RoboDK station: SandBox_RS003N.rdk

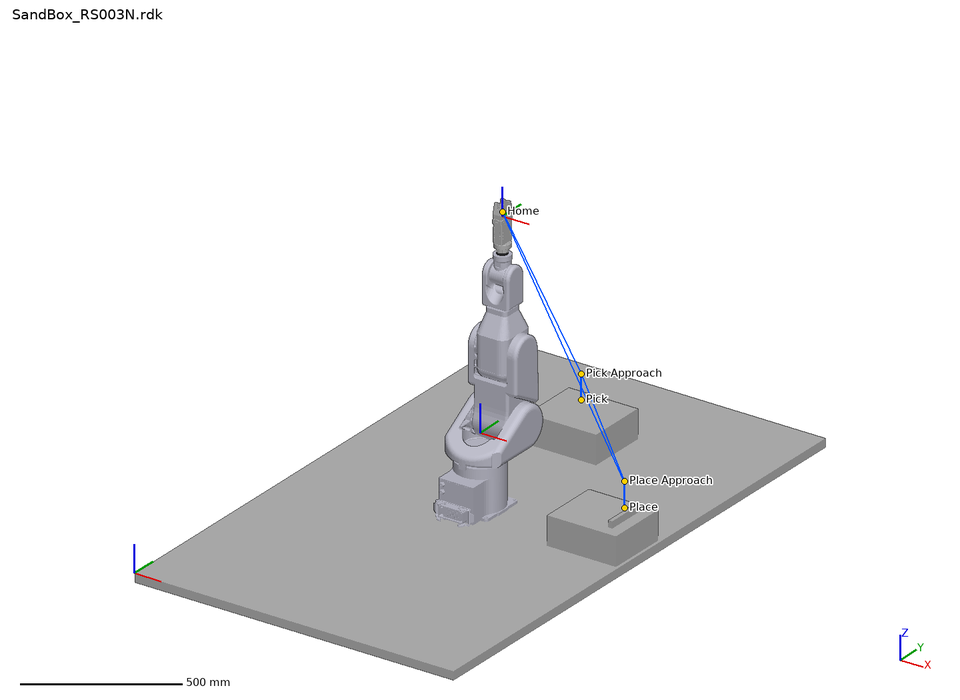
[picture v0: the station drawn from its stored meshes, robots at their saved joint values, targets as dots, program paths as lines]
Station SandBox_RS003N (saved by RoboDK 5.6.1). Poses are relative to the parent item; angles as X-Y-Z fixed-axis rotations.
Station parameters (name, value as stored): Gripper, 6
  - frame Kawasaki RS03N Base at (0, 0, 250) mm
    - robot Kawasaki RS03N: 6 axes, payload 3 kg, reach 620 mm, repeatability 0.02 mm, weight 20 kg
        modified DH rows (alpha deg, a mm, theta deg, d mm): 0, 0, 0, 250; -90, 120, -90, 0; 0, 250, -90, 0; -90, 0, 0, 250; 90, 0, 0, 0; -90, 0, 180, 80
        base shift (0, 0, -250) mm, rotated rx 0 ry 0 rz 90 deg
        joint limits [-160, -60, -150, -360, -135, -360] to [160, 150, 120, 360, 135, 360]; home [0, 0, -90, 0, 0, 0]; saved at [0, 0, 0, 0, 0, 0]
      - tool gripper, TCP at (0, 0, 130) mm, size 79.7 x 56.4 x 121.3 mm, geometry from gripper.stl
      - frame Finger Ref at (0, 0, 115) mm
        - object Finger A at (0, -6, 0) mm, size 21.4 x 34 x 50 mm, geometry from finger.stl
        - object Finger B at (0, 6, 0) mm, size 21.4 x 34 x 50 mm, geometry from finger.stl
    - frame Table2 at (-600, -1000, -250) mm
      - object table at (600, 1000, -30) mm, size 2000 x 1200 x 30 mm, geometry from table.stl
      - target Home (Cartesian target) at (600, 1120, 960) mm; joints [0, 0, 0, 0, 0, 0] of Kawasaki RS03N
      - target Pick Approach (Cartesian target) at (600, 1542.98, 235) mm, rotated rx 180 ry 0 rz 0 deg; joints [0, 43.925, -42.649, 0, -93.426, 0] of Kawasaki RS03N
      - target Pick (Cartesian target) at (600, 1542.98, 145) mm, rotated rx 180 ry 0 rz 0 deg; joints [0, 46.709, -58.7, 0, -74.591, 0] of Kawasaki RS03N
      - target Place Approach (Cartesian target) at (1143.05, 1000, 235) mm, rotated rx -180 ry 0 rz -90 deg; joints [90, 43.948, -42.611, 0, -93.441, 0] of Kawasaki RS03N
      - target Place (Cartesian target) at (1143.05, 1000, 145) mm, rotated rx -180 ry 0 rz -90 deg; joints [90, 46.726, -58.67, 0, -74.604, 0] of Kawasaki RS03N
      - object box at (600, 1550, 0) mm, size 260 x 225 x 105 mm, geometry from box.stl
      - object box2 at (1060, 1000, 0) mm, size 260 x 225 x 105 mm, geometry from box.stl
      - object part at (1150.07, 1000, 118) mm, rotated rx 0 ry 0 rz -90 deg, size 150 x 25 x 15 mm, geometry from part.stl
  - Python program Gripper_RS003N (listed below)
  - program GripperClose (3 instructions, listed below)
  - program GripperOpen (3 instructions, listed below)
  - program ResetSimulation (2 instructions, listed below)
  - program Main (14 instructions, listed below)
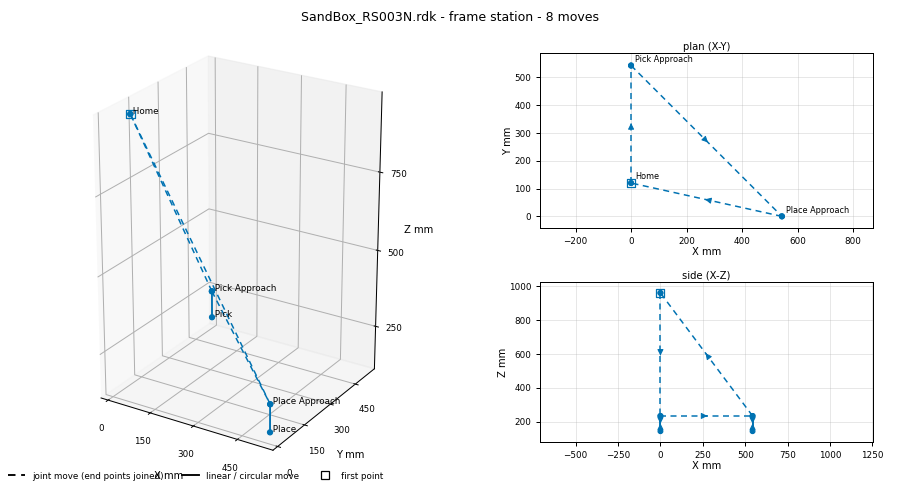
[picture p0: tool path of SandBox_RS003N.rdk in frame station, 8 of 8 moves have a stored position in this frame; points joined in program order, loops and branches not executed]

--- Python program Gripper_RS003N ---
# This program allows moving gripper fingers
import sys # allows getting the passed argument parameters
from robodk import *

if len(sys.argv) < 2:
    print('Invalid parameters. This function must be called as MoveGripper(Gripper_Id, Distance)')
    print('Number of arguments: ' + str(len(sys.argv)))
    #raise Exception('Invalid parameters provided: ' + str(sys.argv))
    entry = mbox('Move gripper. Type:\n1 to open, 0 to close\n\nNote: this can be called as a program.\nExample: Gripper(1)', entry='0')
    if not entry:
        raise Exception('Operation cancelled by user')

    GRIPPER_VALUE = int(entry)*6

else:
    GRIPPER_VALUE = int(sys.argv[1])*6

from robolink import *    # API to communicate with RoboDK
RDK = Robolink()


finger_P = RDK.Item('Finger B')
finger_N = RDK.Item('Finger A')

if not finger_P.Valid() or not finger_N.Valid():
    raise Exception('Invalid Gripper ID')

finger_P.setPose(transl(0,+GRIPPER_VALUE,0))
finger_N.setPose(transl(0,-GRIPPER_VALUE,0))

# Set the station parameter
RDK.setParam('Gripper', GRIPPER_VALUE)

--- program GripperClose (robot Kawasaki RS03N) ---
  Appel Gripper_RS003N(0)
  Attacher à gripper
  Pause 500 ms

--- program GripperOpen (robot Kawasaki RS03N) ---
  Appel Gripper_RS003N(1)
  Détachez de gripper
  Pause 500 ms

--- program ResetSimulation (robot Kawasaki RS03N) ---
  Replacer objets
  Remplacer part

--- program Main (robot Kawasaki RS03N) ---
  Appel ResetSimulation
  Définir Ref.: Table2
  Choisir Outil: gripper
  Appel GripperOpen
  MoveJ (Home)
  MoveJ (Pick Approach)
  MoveL (Pick)
  Appel GripperClose
  MoveL (Pick Approach)
  MoveJ (Place Approach)
  MoveL (Place)
  Appel GripperOpen
  MoveL (Place Approach)
  MoveJ (Home)
